KUKA KRL program: wkz3_ab.src, wkz3_ab.dat

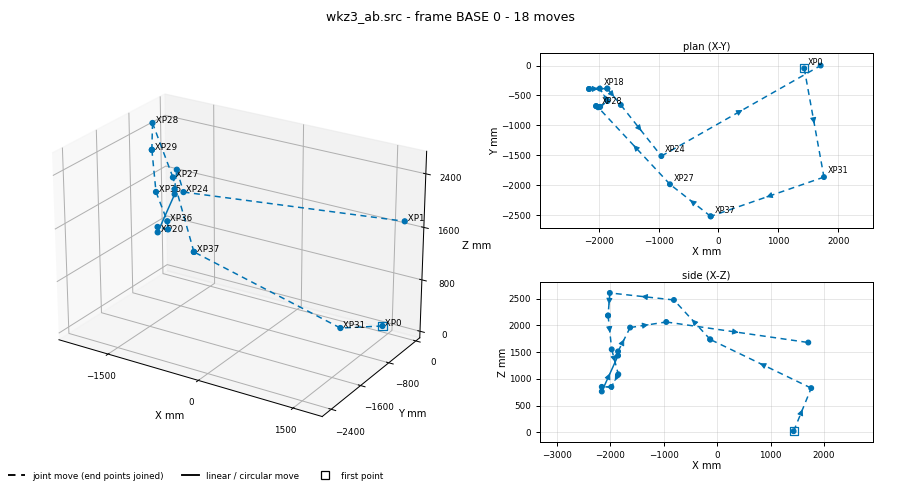
[picture p0: tool path of wkz3_ab.src in frame BASE 0, 18 of 18 moves have a stored position in this frame; points joined in program order, loops and branches not executed]
--- wkz3_ab.src ---
&ACCESS RVO7
&REL 39
&COMMENT Deposito GUN C2
&PARAM DISKPATH = KRC:\R1\Program
DEF wkz3_ab( )
;FOLD INI
  ;FOLD BASISTECH INI
    GLOBAL INTERRUPT DECL 3 WHEN $STOPMESS==TRUE DO IR_STOPM ( )
    INTERRUPT ON 3
    BAS (#INITMOV,0 )
  ;ENDFOLD (BASISTECH INI)
;FOLD GRIPPERTECH INI
USER_GRP(0,DUMMY,DUMMY,GDEFAULT)
;ENDFOLD (GRIPPERTECH INI)
  ;FOLD USER INI
    ;Make your modifications here

  ;ENDFOLD (USER INI)
;ENDFOLD (INI)

; Caracterização dos meios de produção:
; CHANGES: Deposita Pinça C2
; Versão Atual: 18/12/2015
; Name: P13.050-R5

chk_w3_wechs_ok ( )      ; CHECK PINCA C2

;FOLD PTP P0 CONT Vel=100 % PDAT0 Tool[8]:Tool Changer Base[0];%{PE}%R 8.2.20,%MKUKATPBASIS,%CMOVE,%VPTP,%P 1:PTP, 2:P0, 3:C_DIS, 5:100, 7:PDAT0
$BWDSTART=FALSE
PDAT_ACT=PPDAT0
FDAT_ACT=FP0
BAS(#PTP_PARAMS,100)
PTP XP0 C_DIS
;ENDFOLD
;FOLD PTP P31 CONT Vel=100 % PDAT25 Tool[8]:Tool Changer Base[0];%{PE}%R 8.2.20,%MKUKATPBASIS,%CMOVE,%VPTP,%P 1:PTP, 2:P31, 3:C_DIS, 5:100, 7:PDAT25
$BWDSTART=FALSE
PDAT_ACT=PPDAT25
FDAT_ACT=FP31
BAS(#PTP_PARAMS,100)
PTP XP31 C_DIS
;ENDFOLD
;FOLD PTP P37 CONT Vel=100 % PDAT31 Tool[8]:Tool Changer Base[0];%{PE}%R 8.2.20,%MKUKATPBASIS,%CMOVE,%VPTP,%P 1:PTP, 2:P37, 3:C_DIS, 5:100, 7:PDAT31
$BWDSTART=FALSE
PDAT_ACT=PPDAT31
FDAT_ACT=FP37
BAS(#PTP_PARAMS,100)
PTP XP37 C_DIS
;ENDFOLD

if FraesAnf (3) then
;f_fraes3 ()
endif

;FOLD PTP P38 CONT Vel=100 % PDAT32 Tool[8]:Tool Changer Base[0];%{PE}%R 8.2.20,%MKUKATPBASIS,%CMOVE,%VPTP,%P 1:PTP, 2:P38, 3:C_DIS, 5:100, 7:PDAT32
$BWDSTART=FALSE
PDAT_ACT=PPDAT32
FDAT_ACT=FP38
BAS(#PTP_PARAMS,100)
PTP XP38 C_DIS
;ENDFOLD
;FOLD PTP P27 CONT Vel=100 % PDAT21 Tool[8]:Tool Changer Base[0];%{PE}%R 8.2.20,%MKUKATPBASIS,%CMOVE,%VPTP,%P 1:PTP, 2:P27, 3:C_DIS, 5:100, 7:PDAT21
$BWDSTART=FALSE
PDAT_ACT=PPDAT21
FDAT_ACT=FP27
BAS(#PTP_PARAMS,100)
PTP XP27 C_DIS
;ENDFOLD

;FOLD PULSE 192 'DOCK 4 Fechar Proteção' State=TRUE CONT Time=1 sec;%{PE}%R 8.2.20,%MKUKATPBASIS,%COUT,%VPULSE,%P 2:192, 3:DOCK 4 Fechar Proteção, 5:TRUE, 6:CONTINUE, 8:1
CONTINUE
PULSE($OUT[192], TRUE,1)
;ENDFOLD
;FOLD WAIT FOR NOT ( IN 189 'DOCK 4 Proteção Aberta' ) CONT;%{PE}%R 8.2.20,%MKUKATPBASIS,%CEXT_WAIT_FOR,%VEXT_WAIT_FOR,%P 2:NOT, 4:, 5:$IN, 6:189, 7:DOCK 4 Proteção Aberta, 9:CONTINUE
CONTINUE
WAIT FOR  NOT ( $IN[189] )
;ENDFOLD
;FOLD WAIT FOR ( IN 190 'DOCK 4 Proteção Fechada' ) CONT;%{PE}%R 8.2.20,%MKUKATPBASIS,%CEXT_WAIT_FOR,%VEXT_WAIT_FOR,%P 2:, 4:, 5:$IN, 6:190, 7:DOCK 4 Proteção Fechada, 9:CONTINUE
CONTINUE
WAIT FOR  ( $IN[190] )
;ENDFOLD

;FOLD PTP P28 CONT Vel=100 % PDAT22 Tool[8]:Tool Changer Base[0];%{PE}%R 8.2.20,%MKUKATPBASIS,%CMOVE,%VPTP,%P 1:PTP, 2:P28, 3:C_DIS, 5:100, 7:PDAT22
$BWDSTART=FALSE
PDAT_ACT=PPDAT22
FDAT_ACT=FP28
BAS(#PTP_PARAMS,100)
PTP XP28 C_DIS
;ENDFOLD
;FOLD PTP P29 CONT Vel=100 % PDAT23 Tool[8]:Tool Changer Base[0];%{PE}%R 8.2.20,%MKUKATPBASIS,%CMOVE,%VPTP,%P 1:PTP, 2:P29, 3:C_DIS, 5:100, 7:PDAT23
$BWDSTART=FALSE
PDAT_ACT=PPDAT23
FDAT_ACT=FP29
BAS(#PTP_PARAMS,100)
PTP XP29 C_DIS
;ENDFOLD
;FOLD PTP P26 CONT Vel=100 % PDAT20 Tool[8]:Tool Changer Base[0];%{PE}%R 8.2.20,%MKUKATPBASIS,%CMOVE,%VPTP,%P 1:PTP, 2:P26, 3:C_DIS, 5:100, 7:PDAT20
$BWDSTART=FALSE
PDAT_ACT=PPDAT20
FDAT_ACT=FP26
BAS(#PTP_PARAMS,100)
PTP XP26 C_DIS
;ENDFOLD

;FOLD WAIT FOR ( NOT IN 169 'DOCK 2 Deposito Ocupado' ) CONT;%{PE}%R 8.2.20,%MKUKATPBASIS,%CEXT_WAIT_FOR,%VEXT_WAIT_FOR,%P 2:, 4:NOT, 5:$IN, 6:169, 7:DOCK 2 Deposito Ocupado, 9:CONTINUE
CONTINUE
WAIT FOR  (  NOT $IN[169] )
;ENDFOLD
;FOLD WAIT FOR ( IN 219 'Posicao p/ Acoplamento OK' ) CONT;%{PE}%R 8.2.20,%MKUKATPBASIS,%CEXT_WAIT_FOR,%VEXT_WAIT_FOR,%P 2:, 4:, 5:$IN, 6:219, 7:Posicao p/ Acoplamento OK, 9:CONTINUE
CONTINUE
WAIT FOR  ( $IN[219] )
;ENDFOLD
;FOLD PULSE 175 'DOCK 2 Abrir Proteção' State=TRUE CONT Time=1 sec;%{PE}%R 8.2.20,%MKUKATPBASIS,%COUT,%VPULSE,%P 2:175, 3:DOCK 2 Abrir Proteção, 5:TRUE, 6:CONTINUE, 8:1
CONTINUE
PULSE($OUT[175], TRUE,1)
;ENDFOLD
;FOLD WAIT FOR ( IN 173 'DOCK 2 Proteção Aberta' ) CONT;%{PE}%R 8.2.20,%MKUKATPBASIS,%CEXT_WAIT_FOR,%VEXT_WAIT_FOR,%P 2:, 4:, 5:$IN, 6:173, 7:DOCK 2 Proteção Aberta, 9:CONTINUE
CONTINUE
WAIT FOR  ( $IN[173] )
;ENDFOLD
;FOLD WAIT FOR NOT ( IN 174 'DOCK 2 Proteção Fechada' ) CONT;%{PE}%R 8.2.20,%MKUKATPBASIS,%CEXT_WAIT_FOR,%VEXT_WAIT_FOR,%P 2:NOT, 4:, 5:$IN, 6:174, 7:DOCK 2 Proteção Fechada, 9:CONTINUE
CONTINUE
WAIT FOR  NOT ( $IN[174] )
;ENDFOLD

;FOLD PTP P35 CONT Vel=100 % PDAT29 Tool[8]:Tool Changer Base[0];%{PE}%R 8.2.20,%MKUKATPBASIS,%CMOVE,%VPTP,%P 1:PTP, 2:P35, 3:C_DIS, 5:100, 7:PDAT29
$BWDSTART=FALSE
PDAT_ACT=PPDAT29
FDAT_ACT=FP35
BAS(#PTP_PARAMS,100)
PTP XP35 C_DIS
;ENDFOLD
;FOLD PTP P36 CONT Vel=100 % PDAT30 Tool[8]:Tool Changer Base[0];%{PE}%R 8.2.20,%MKUKATPBASIS,%CMOVE,%VPTP,%P 1:PTP, 2:P36, 3:C_DIS, 5:100, 7:PDAT30
$BWDSTART=FALSE
PDAT_ACT=PPDAT30
FDAT_ACT=FP36
BAS(#PTP_PARAMS,100)
PTP XP36 C_DIS
;ENDFOLD
;FOLD PTP P18 CONT Vel=100 % PDAT15 Tool[8]:Tool Changer Base[0];%{PE}%R 8.2.20,%MKUKATPBASIS,%CMOVE,%VPTP,%P 1:PTP, 2:P18, 3:C_DIS, 5:100, 7:PDAT15
$BWDSTART=FALSE
PDAT_ACT=PPDAT15
FDAT_ACT=FP18
BAS(#PTP_PARAMS,100)
PTP XP18 C_DIS
;ENDFOLD
;FOLD PTP P19 Vel=100 % PDAT16 Tool[3]:Gun C2 Base[0];%{PE}%R 8.2.20,%MKUKATPBASIS,%CMOVE,%VPTP,%P 1:PTP, 2:P19, 3:, 5:100, 7:PDAT16
$BWDSTART=FALSE
PDAT_ACT=PPDAT16
FDAT_ACT=FP19
BAS(#PTP_PARAMS,100)
PTP XP19
;ENDFOLD

;FOLD ; ponto de deposito da ferramenta;%{PE}%R 8.2.19,%MKUKATPBASIS,%CCOMMENT,%VNORMAL,%P 2:ponto  de  deposito  da  ferramenta
;ENDFOLD
;FOLD LIN P20 Vel=0.1 m/s CPDAT6 Tool[3]:Gun C2 Base[0];%{PE}%R 8.2.20,%MKUKATPBASIS,%CMOVE,%VLIN,%P 1:LIN, 2:P20, 3:, 5:0.1, 7:CPDAT6
$BWDSTART=FALSE
LDAT_ACT=LCPDAT6
FDAT_ACT=FP20
BAS(#CP_PARAMS,0.1)
LIN XP20
;ENDFOLD

;FOLD WAIT Time=0.5 sec;%{PE}%R 8.2.20,%MKUKATPBASIS,%CWAIT,%VWAIT,%P 3:0.5
WAIT SEC 0.5
;ENDFOLD
;FOLD WAIT FOR ( IN 169 'DOCK 2 Deposito Ocupado' );%{PE}%R 8.2.20,%MKUKATPBASIS,%CEXT_WAIT_FOR,%VEXT_WAIT_FOR,%P 2:, 4:, 5:$IN, 6:169, 7:DOCK 2 Deposito Ocupado, 9:
WAIT FOR  ( $IN[169] )
;ENDFOLD
;FOLD OUT 224 'Bloquear MPS' State=FALSE ;%{PE}%R 8.2.20,%MKUKATPBASIS,%COUT,%VOUTX,%P 2:224, 3:Bloquear MPS, 5:FALSE, 6:
$OUT[224]=FALSE
;ENDFOLD
;FOLD OUT 223 'Desbloquear MPS' State=TRUE ;%{PE}%R 8.2.20,%MKUKATPBASIS,%COUT,%VOUTX,%P 2:223, 3:Desbloquear MPS, 5:TRUE, 6:
$OUT[223]=TRUE
;ENDFOLD
;FOLD WAIT FOR ( IN 217 'MPS Destravado' );%{PE}%R 8.2.20,%MKUKATPBASIS,%CEXT_WAIT_FOR,%VEXT_WAIT_FOR,%P 2:, 4:, 5:$IN, 6:217, 7:MPS Destravado, 9:
WAIT FOR  ( $IN[217] )
;ENDFOLD
;FOLD WAIT FOR ( NOT IN 221 'MPS Travado' );%{PE}%R 8.2.20,%MKUKATPBASIS,%CEXT_WAIT_FOR,%VEXT_WAIT_FOR,%P 2:, 4:NOT, 5:$IN, 6:221, 7:MPS Travado, 9:
WAIT FOR  (  NOT $IN[221] )
;ENDFOLD
;FOLD IBUS OFF;%{PE}%R 8.2.20,%MKUKATPBASIS,%CIBUS,%VMAP,%P 2:#OFF, 3:1
$IBUS_OFF=$IBUS_ON
$IBUS_ON=0
;ENDFOLD
;FOLD WAIT Time=0.5 sec;%{PE}%R 8.2.20,%MKUKATPBASIS,%CWAIT,%VWAIT,%P 3:0.5
WAIT SEC 0.5
;ENDFOLD

;FOLD LIN P25 Vel=0.1 m/s CPDAT8 Tool[8]:Tool Changer Base[0];%{PE}%R 8.2.20,%MKUKATPBASIS,%CMOVE,%VLIN,%P 1:LIN, 2:P25, 3:, 5:0.1, 7:CPDAT8
$BWDSTART=FALSE
LDAT_ACT=LCPDAT8
FDAT_ACT=FP25
BAS(#CP_PARAMS,0.1)
LIN XP25
;ENDFOLD
;FOLD LIN P21 CONT Vel=1 m/s CPDAT7 Tool[8]:Tool Changer Base[0];%{PE}%R 8.2.20,%MKUKATPBASIS,%CMOVE,%VLIN,%P 1:LIN, 2:P21, 3:C_DIS C_DIS, 5:1, 7:CPDAT7
$BWDSTART=FALSE
LDAT_ACT=LCPDAT7
FDAT_ACT=FP21
BAS(#CP_PARAMS,1)
LIN XP21 C_DIS C_DIS
;ENDFOLD

;FOLD WAIT FOR ( IN 169 'DOCK 2 Deposito Ocupado' ) CONT;%{PE}%R 8.2.20,%MKUKATPBASIS,%CEXT_WAIT_FOR,%VEXT_WAIT_FOR,%P 2:, 4:, 5:$IN, 6:169, 7:DOCK 2 Deposito Ocupado, 9:CONTINUE
CONTINUE
WAIT FOR  ( $IN[169] )
;ENDFOLD
;FOLD WAIT FOR ( NOT IN 219 'Posicao p/ Acoplamento OK' ) CONT;%{PE}%R 8.2.20,%MKUKATPBASIS,%CEXT_WAIT_FOR,%VEXT_WAIT_FOR,%P 2:, 4:NOT, 5:$IN, 6:219, 7:Posicao p/ Acoplamento OK, 9:CONTINUE
CONTINUE
WAIT FOR  (  NOT $IN[219] )
;ENDFOLD
;FOLD OUT 223 'Desbloquear MPS' State=FALSE CONT;%{PE}%R 8.2.20,%MKUKATPBASIS,%COUT,%VOUTX,%P 2:223, 3:Desbloquear MPS, 5:FALSE, 6:CONTINUE
CONTINUE
$OUT[223]=FALSE
;ENDFOLD
;FOLD WAIT FOR NOT ( IN 189 'DOCK 4 Proteção Aberta' ) CONT;%{PE}%R 8.2.20,%MKUKATPBASIS,%CEXT_WAIT_FOR,%VEXT_WAIT_FOR,%P 2:NOT, 4:, 5:$IN, 6:189, 7:DOCK 4 Proteção Aberta, 9:CONTINUE
CONTINUE
WAIT FOR  NOT ( $IN[189] )
;ENDFOLD
;FOLD WAIT FOR ( IN 190 'DOCK 4 Proteção Fechada' ) CONT;%{PE}%R 8.2.20,%MKUKATPBASIS,%CEXT_WAIT_FOR,%VEXT_WAIT_FOR,%P 2:, 4:, 5:$IN, 6:190, 7:DOCK 4 Proteção Fechada, 9:CONTINUE
CONTINUE
WAIT FOR  ( $IN[190] )
;ENDFOLD

;FOLD PTP P22 CONT Vel=100 % PDAT17 Tool[8]:Tool Changer Base[0];%{PE}%R 8.2.20,%MKUKATPBASIS,%CMOVE,%VPTP,%P 1:PTP, 2:P22, 3:C_DIS, 5:100, 7:PDAT17
$BWDSTART=FALSE
PDAT_ACT=PPDAT17
FDAT_ACT=FP22
BAS(#PTP_PARAMS,100)
PTP XP22 C_DIS
;ENDFOLD
;FOLD PTP P24 CONT Vel=100 % PDAT19 Tool[8]:Tool Changer Base[0];%{PE}%R 8.2.20,%MKUKATPBASIS,%CMOVE,%VPTP,%P 1:PTP, 2:P24, 3:C_DIS, 5:100, 7:PDAT19
$BWDSTART=FALSE
PDAT_ACT=PPDAT19
FDAT_ACT=FP24
BAS(#PTP_PARAMS,100)
PTP XP24 C_DIS
;ENDFOLD
;FOLD PTP P1 CONT Vel=100 % PDAT1 Tool[8]:Tool Changer Base[0];%{PE}%R 8.2.20,%MKUKATPBASIS,%CMOVE,%VPTP,%P 1:PTP, 2:P1, 3:C_DIS, 5:100, 7:PDAT1
$BWDSTART=FALSE
PDAT_ACT=PPDAT1
FDAT_ACT=FP1
BAS(#PTP_PARAMS,100)
PTP XP1 C_DIS
;ENDFOLD

;FOLD PULSE 176 'DOCK 2 Fechar Proteção' State=TRUE Time=1 sec;%{PE}%R 8.2.20,%MKUKATPBASIS,%COUT,%VPULSE,%P 2:176, 3:DOCK 2 Fechar Proteção, 5:TRUE, 6:, 8:1
PULSE($OUT[176], TRUE,1)
;ENDFOLD

END

--- wkz3_ab.dat ---
&ACCESS RVO7
&REL 39
&COMMENT Deposito GUN C2
&PARAM DISKPATH = KRC:\R1\Program
DEFDAT  wkz3_ab
;FOLD EXTERNAL DECLARATIONS;%{PE}%MKUKATPBASIS,%CEXT,%VCOMMON,%P
;FOLD GRIPPERTECH EXT
EXT  H50 (INT  :IN,INT  :IN,INT  :IN,GRP_TYP  :IN )
;ENDFOLD (GRIPPERTECH EXT)
;FOLD SPOTTECH EXT
EXT  USERSPOT (S_COMMAND  :IN,SPOT_TYPE  :IN )
;ENDFOLD (SPOTTECH EXT)
;FOLD BASISTECH EXT;%{PE}%MKUKATPBASIS,%CEXT,%VEXT,%P
EXT  BAS (BAS_COMMAND  :IN,REAL  :IN )
DECL INT SUCCESS
;ENDFOLD (BASISTECH EXT)
;FOLD USER EXT;%{E}%MKUKATPUSER,%CEXT,%VEXT,%P
;Make your modifications here

;ENDFOLD (USER EXT)
;ENDFOLD (EXTERNAL DECLARATIONS)
;# ============ START PATH : zax_p13050r5_02 =============
DECL BASIS_SUGG_T LAST_BASIS={POINT1[] "P1                      ",POINT2[] "P1                      ",CP_PARAMS[] "CPDAT0                  ",PTP_PARAMS[] "PDAT1                   ",CONT[] "C_DIS                   ",CP_VEL[] "2.0                     ",PTP_VEL[] "100                     ",SYNC_PARAMS[] "SYNCDAT                 ",SPL_NAME[] "S0                      "}
DECL PDAT PPDAT15={VEL 100.0,ACC 100.0,APO_DIST 50.0,APO_MODE #CDIS}
DECL E6POS XP18={X -1983.39905,Y -384.658997,Z 848.571899,A 179.405396,B -20.0995808,C 0.287330389,S 2,T 2,E1 0.0,E2 0.0,E3 0.0,E4 0.0,E5 0.0,E6 0.0}
DECL FDAT FP18={TOOL_NO 3,BASE_NO 0,IPO_FRAME #BASE,POINT2[] " ",TQ_STATE FALSE}
DECL PDAT PPDAT16={VEL 100.0,ACC 100.0,APO_DIST 0.0,APO_MODE #CDIS}
DECL E6POS XP19={X -2163.06299,Y -391.910309,Z 849.493713,A 179.144699,B -15.9372597,C 0.885988176,S 2,T 10,E1 0.0,E2 0.0,E3 0.0,E4 0.0,E5 0.0,E6 0.0}
DECL FDAT FP19={TOOL_NO 3,BASE_NO 0,IPO_FRAME #BASE,POINT2[] " ",TQ_STATE FALSE}
DECL LDAT LCPDAT6={VEL 2.0,ACC 100.0,APO_DIST 100.0,APO_FAC 50.0,AXIS_VEL 100.0,AXIS_ACC 100.0,ORI_TYP #VAR,CIRC_TYP #BASE,JERK_FAC 50.0,GEAR_JERK 50.0,EXAX_IGN 0}
DECL E6POS XP20={X -2162.98901,Y -391.650299,Z 762.729614,A 179.142395,B -15.9539003,C 0.890016377,S 2,T 10,E1 0.0,E2 0.0,E3 0.0,E4 0.0,E5 0.0,E6 0.0}
DECL FDAT FP20={TOOL_NO 3,BASE_NO 0,IPO_FRAME #BASE,POINT2[] " ",TQ_STATE FALSE}
DECL LDAT LCPDAT7={VEL 2.0,ACC 100.0,APO_DIST 100.0,APO_FAC 50.0,AXIS_VEL 100.0,AXIS_ACC 100.0,ORI_TYP #VAR,CIRC_TYP #BASE,JERK_FAC 50.0,GEAR_JERK 50.0,EXAX_IGN 0}
DECL E6POS XP21={X -1857.92102,Y -385.258209,Z 1513.73303,A -165.6259,B -1.12822604,C -179.4198,S 2,T 10,E1 0.0,E2 0.0,E3 0.0,E4 0.0,E5 0.0,E6 0.0}
DECL FDAT FP21={TOOL_NO 8,BASE_NO 0,IPO_FRAME #BASE,POINT2[] " ",TQ_STATE FALSE}
DECL PDAT PPDAT17={VEL 100.0,ACC 100.0,APO_DIST 100.0,APO_MODE #CDIS}
DECL E6POS XP22={X -1632.07996,Y -659.100586,Z 1960.99597,A -152.860703,B -43.9183006,C 177.1689,S 2,T 10,E1 0.0,E2 0.0,E3 0.0,E4 0.0,E5 0.0,E6 0.0}
DECL FDAT FP22={TOOL_NO 8,BASE_NO 0,IPO_FRAME #BASE,POINT2[] " ",TQ_STATE FALSE}
DECL PDAT PPDAT19={VEL 100.0,ACC 100.0,APO_DIST 100.0,APO_MODE #CDIS}
DECL E6POS XP24={X -955.036621,Y -1513.44702,Z 2065.44092,A -167.067596,B -36.9554291,C -148.494507,S 2,T 10,E1 0.0,E2 0.0,E3 0.0,E4 0.0,E5 0.0,E6 0.0}
DECL FDAT FP24={TOOL_NO 8,BASE_NO 0,IPO_FRAME #BASE,POINT2[] " ",TQ_STATE FALSE}
DECL E6POS XP25={X -1857.96997,Y -385.265198,Z 1435.11804,A -165.625595,B -1.13914704,C -179.420395,S 2,T 10,E1 0.0,E2 0.0,E3 0.0,E4 0.0,E5 0.0,E6 0.0}
DECL FDAT FP25={TOOL_NO 8,BASE_NO 0,IPO_FRAME #BASE,POINT2[] " ",TQ_STATE FALSE}
DECL LDAT LCPDAT8={VEL 2.0,ACC 100.0,APO_DIST 100.0,APO_FAC 50.0,AXIS_VEL 100.0,AXIS_ACC 100.0,ORI_TYP #VAR,CIRC_TYP #BASE,JERK_FAC 50.0,GEAR_JERK 50.0,EXAX_IGN 0}
DECL E6POS XP26={X -2044.98596,Y -678.077515,Z 2186.08789,A 128.082397,B -61.4635811,C 56.5986595,S 2,T 2,E1 0.0,E2 0.0,E3 0.0,E4 0.0,E5 0.0,E6 0.0}
DECL FDAT FP26={TOOL_NO 3,BASE_NO 0,IPO_FRAME #BASE,POINT2[] " ",TQ_STATE FALSE}
DECL PDAT PPDAT20={VEL 100.0,ACC 100.0,APO_DIST 50.0,APO_MODE #CDIS}
DECL PDAT PPDAT21={VEL 100.0,ACC 100.0,APO_DIST 0.0,APO_MODE #CDIS}
DECL E6POS XP27={X -811.198486,Y -1984.42798,Z 2477.93408,A 142.229599,B -34.2021408,C 95.1900864,S 2,T 2,E1 0.0,E2 0.0,E3 0.0,E4 0.0,E5 0.0,E6 0.0}
DECL FDAT FP27={TOOL_NO 3,BASE_NO 0,IPO_FRAME #BASE,POINT2[] " ",TQ_STATE FALSE}
DECL PDAT PPDAT22={VEL 100.0,ACC 100.0,APO_DIST 100.0,APO_MODE #CDIS}
DECL E6POS XP28={X -2012.125,Y -697.976013,Z 2609.73901,A 86.4610291,B -54.3633003,C 105.463097,S 2,T 2,E1 0.0,E2 0.0,E3 0.0,E4 0.0,E5 0.0,E6 0.0}
DECL FDAT FP28={TOOL_NO 3,BASE_NO 0,IPO_FRAME #BASE,POINT2[] " ",TQ_STATE FALSE}
DECL PDAT PPDAT23={VEL 100.0,ACC 100.0,APO_DIST 100.0,APO_MODE #CDIS}
DECL E6POS XP29={X -2045.06006,Y -678.063293,Z 2186.052,A 128.084702,B -61.4636307,C 56.5944786,S 2,T 2,E1 0.0,E2 0.0,E3 0.0,E4 0.0,E5 0.0,E6 0.0}
DECL FDAT FP29={TOOL_NO 3,BASE_NO 0,IPO_FRAME #BASE,POINT2[] " ",TQ_STATE FALSE}
DECL E6POS XP31={X 1762.06995,Y -1864.10596,Z 826.058289,A 157.848907,B 46.1915894,C 35.5948105,S 6,T 26,E1 0.0,E2 0.0,E3 0.0,E4 0.0,E5 0.0,E6 0.0}
DECL FDAT FP31={TOOL_NO 3,BASE_NO 0,IPO_FRAME #BASE,POINT2[] " ",TQ_STATE FALSE}
DECL PDAT PPDAT25={VEL 100.0,ACC 100.0,APO_DIST 100.0,APO_MODE #CDIS}
DECL SPOT_SUGG_T LAST_SPOT={GUN[] "3                       ",RETR_CMD[] "#OPN                    ",CHOISE[] "#FIRST                  ",CLO_TM[] "1                       ",PGNO1[] "171                     ",PRESS1[] "0                       ",PGNO2[] "1                       ",PRESS2[] "0                       ",SPOT_PARAMS[] "NORMAL                  "}
DECL E6POS XP35={X -1977.23401,Y -689.853577,Z 1551.77002,A 162.870102,B -51.3725395,C 18.9944096,S 2,T 2,E1 0.0,E2 0.0,E3 0.0,E4 0.0,E5 0.0,E6 0.0}
DECL FDAT FP35={TOOL_NO 3,BASE_NO 0,IPO_FRAME #BASE,POINT2[] " ",TQ_STATE FALSE}
DECL PDAT PPDAT29={VEL 100.0,ACC 100.0,APO_DIST 50.0,APO_MODE #CDIS}
DECL E6POS XP36={X -1853.23901,Y -593.246277,Z 1084.94995,A 179.051498,B -29.9354305,C 1.12474895,S 2,T 2,E1 0.0,E2 0.0,E3 0.0,E4 0.0,E5 0.0,E6 0.0}
DECL FDAT FP36={TOOL_NO 3,BASE_NO 0,IPO_FRAME #BASE,POINT2[] " ",TQ_STATE FALSE}
DECL PDAT PPDAT30={VEL 100.0,ACC 100.0,APO_DIST 50.0,APO_MODE #CDIS}
DECL PDAT PPDAT31={VEL 100.0,ACC 100.0,APO_DIST 100.0,APO_MODE #CDIS}
DECL E6POS XP37={X -130.570404,Y -2520.30103,Z 1737.70203,A 162.716599,B 25.4412403,C 70.1682587,S 2,T 10,E1 0.0,E2 0.0,E3 0.0,E4 0.0,E5 0.0,E6 0.0}
DECL FDAT FP37={TOOL_NO 3,BASE_NO 0,IPO_FRAME #BASE,POINT2[] " ",TQ_STATE FALSE}
DECL PDAT PPDAT32={VEL 100.0,ACC 100.0,APO_DIST 100.0,APO_MODE #CDIS}
DECL E6POS XP38={X -130.568695,Y -2520.29907,Z 1737.70398,A 162.716705,B 25.4413395,C 70.1683273,S 2,T 10,E1 0.0,E2 0.0,E3 0.0,E4 0.0,E5 0.0,E6 0.0}
DECL FDAT FP38={TOOL_NO 3,BASE_NO 0,IPO_FRAME #BASE,POINT2[] " ",TQ_STATE FALSE}
DECL E6POS XP39={X 1286.59497,Y -1367.25098,Z 2703.1709,A -0.3803339,B 45.2661896,C -42.7513695,S 2,T 2,E1 0.0,E2 0.0,E3 0.0,E4 0.0,E5 0.0,E6 0.0}
DECL FDAT FP39={TOOL_NO 9,BASE_NO 3,IPO_FRAME #BASE,POINT2[] " ",TQ_STATE FALSE}
DECL PDAT PPDAT33={VEL 100.0,ACC 100.0,APO_DIST 100.0}
DECL PDAT PPDAT0={VEL 100.0,ACC 100.0,APO_DIST 100.0,APO_MODE #CDIS}
DECL E6POS XP0={X 1432.48596,Y -47.8588409,Z 18.4852104,A 172.328903,B -14.6202898,C -2.31678104,S 6,T 26,E1 0.0,E2 0.0,E3 0.0,E4 0.0,E5 0.0,E6 0.0}
DECL FDAT FP0={TOOL_NO 3,BASE_NO 0,IPO_FRAME #BASE,POINT2[] " ",TQ_STATE FALSE}
DECL E6POS XP1={X 1707.34802,Y -0.0147145698,Z 1680.53003,A -76.93647,B -7.43512583,C -150.8535,S 2,T 2,E1 0.0,E2 0.0,E3 0.0,E4 0.0,E5 0.0,E6 0.0}
DECL FDAT FP1={TOOL_NO 8,BASE_NO 0,IPO_FRAME #BASE,POINT2[] " ",TQ_STATE FALSE}
DECL PDAT PPDAT1={VEL 100.0,ACC 100.0,APO_DIST 100.0,APO_MODE #CDIS}
ENDDAT
